// TIA Portal V20 export
TYPE "UDT_EmisionDeMesa"
   STRUCT
      Auxiliar_01 : UInt;
      Auxiliar_02 : UInt;
      Auxiliar_03 : UInt;
      Auxiliar_04 : UInt;
      Protocolo { S7_SetPoint := 'True'} : "UDT_ProtocoloEmiMesa";
   END_STRUCT;
END_TYPE
